DATA_BLOCK "MainDB"
{ S7_Optimized_Access := 'TRUE'; DB_Accessible_From_OPC_UA := 'TRUE'; DB_Accessible_From_Webserver := 'TRUE' }
VERSION : '1.0'
VAR
    LAST_CYCLE_TIME : TIME;
    PROCESS_MATRIX : ARRAY[0..2,0..3] OF "ProcessData_001";
END_VAR

VAR RETAIN
    ALL_TYPES : "TestAllTypes_001";
    CYCLE_COUNT : INT;
    PROCESS_HISTORY : ARRAY[0..9] OF "ProcessData_001";
END_VAR
END_DATA_BLOCK